FUNCTION_BLOCK Pressure EXTENDS SM_Pressure
VAR_INPUT
END_VAR
VAR_OUTPUT
END_VAR
VAR
    _testVar_Pressure : BOOL;
END_VAR

SUPER^();

END_FUNCTION_BLOCK

(* stored: Version 1.1.0.1, ProductVersion 3.1.4018.2
   POU Pressure: Id {ca6f748a-613d-4cab-83f7-833d3799ddc9}, SpecialFunc None *)
